TYPE
  (* Standard: 61499-1 *)
  (* Version 1.0, 2026-07-21, Dimitrios Kalligaridis *)
  PACKAGE mypackage;
  CycleB : STRUCT
    a : mypackage::CycleA;
  END_STRUCT;
END_TYPE
